// TIA Portal V17 export
// export: Created 2025-04-14T03:06:09.7073526Z, ExportSetting WithDefaults, DisplayName Totally Integrated Automation Portal, DisplayVersion V17, DisplayName TIA Portal Openness, DisplayVersion V17, DisplayName TIA Portal Version Control Interface, DisplayVersion V17, DisplayName SINAMICS Startdrive Advanced, DisplayVersion V17, DisplayName SINAMICS Startdrive G130, G150, S120, S150, SINAMICS MV, S210, DisplayVersion V17, DisplayName SINAMICS Startdrive G110M, G120, G120C, G120D, G120P, G115D, DisplayVersion V17, DisplayName STEP 7 Professional, DisplayVersion V17, DisplayName STEP 7 Safety, DisplayVersion V17, DisplayName WinCC Advanced, DisplayVersion V17
TYPE "UDT_Valve_Temp"
// stored: IsFailsafeCompliant false
   STRUCT
      IN_xAutoCmd : Bool;   // 自动模式开阀
      IN_xManualCmd : Bool;   // 手动模式下的阀门控制辅助命令/1为开，0为关
      IN_xOpenCondition : Bool := TRUE;   // 开阀运行条件
      IN_xCloseCondition : Bool := TRUE;   // 关阀运行条件
      OUT_xOpenOK : Bool;   // 开到位
      OUT_xCloseOK : Bool;   // 关到位
   END_STRUCT;
END_TYPE
